FUNCTION TryConvert_BOOL_TO_BYTE : BOOL
VAR_INPUT
	in : BOOL;
	out : REFERENCE TO BYTE;
END_VAR

out := BOOL_TO_BYTE(in);
TryConvert_BOOL_TO_BYTE := TRUE;

END_FUNCTION

(* stored: Version 1.1.0.1, ProductVersion 3.1.4024.12
   POU TryConvert_BOOL_TO_BYTE: Id {d4e08cc2-0d8f-471d-ab77-165a23a10e81}, SpecialFunc None *)
